(* Logix 5000 project; controller DAD143_Test0 1769-L16ER-BB1B rev 34.12; software revision 34.01; part 2 of 2 *)
(* tags used below, declared in another part *)
   CE_Write_Done : BOOL;
   Done_CE : BOOL;
   CE_Start : BOOL;
   Cycle_Start : BOOL;
   DecimalPoint : SINT;
   Display_real : REAL;
   DisplayStr : STRING;
   DP : BOOL;
   DP_Cahr : STRING;
   DP_Read_Par : SINT[3];
   DP_Read_Res : SINT[5];
   DP_Val : SINT;
   DpPos : DINT;
   DS : BOOL;
   DS_Change : BOOL;
   DS_Change_Handshake : BOOL;
   DS_Change_Tag : BOOL;
   DS_Read_Par : SINT[3];
   DS_Read_Res : SINT[5];
   DS_Step1 : BOOL;
   DS_Val : DINT;
   FinalStr : STRING;
   FM_Change : BOOL;
   FM_Change_Handshake : BOOL;
   FM_Change_Tag : BOOL;
   FM_Read_Par : SINT[3];
   FM_Step1 : BOOL;
   FM_Val : SINT;
   gross : BOOL;
   Gross_weight : BOOL;
   Int_reading : BOOL;
   MR : BOOL;
   MR_Change : BOOL;
   MR_Change_Handshake : BOOL;
   MR_Change_Tag : BOOL;
   MR_Read_Par : SINT[3];
   MR_Step1 : BOOL;
   MR_Val : SINT;
   Power_T : TIMER[12];
   Power_T0 : TIMER;
   READ_AOI : AOI_DAD_143_Read[18];
   ReadCDP : MESSAGE;
   ReadDS : MESSAGE;
   Stable_Bit : BOOL;
   Start : BOOL;
   Start_Visibility : BOOL;
   T10 : TIMER;
   T11 : TIMER;
   T12 : TIMER;
   T13 : TIMER;
   T14 : TIMER;
   T15 : TIMER;
   T16 : TIMER;
   T17 : TIMER;
   T18 : TIMER;
   T22 : TIMER;
   T23 : TIMER;
   T24 : TIMER;
   T37 : TIMER;
   T38 : TIMER;
   T39 : TIMER;
   T7 : TIMER;
   T8 : TIMER;
   T9 : TIMER;
   Tare_reset : BOOL;
   Tare_Reset_1 : BOOL;
   Tare_reset_Bit : BOOL;
   Tare_set : BOOL;
   Tare_set_Bit : BOOL;
   TN_Change : BOOL;
   TN_Change_Handshake : BOOL;
   TN_Change_Tag : BOOL;
   TN_Read_Par : SINT[3];
   TN_Step1 : BOOL;
   TN_Val : SINT;
   Write_AOI : AOI_DAD_143_Write[12];
   Write_DS_Par : SINT[7];
   Write_FM_Par : SINT[7];
   Write_MR_Par : SINT[7];
   Write_TN_Par : SINT[7];
   Write_ZI_Par : SINT[7];
   Write_ZN_Par : SINT[7];
   WriteDS : MESSAGE;
   WriteFM : MESSAGE;
   WriteMR : MESSAGE;
   WriteTN : MESSAGE;
   WriteZI : MESSAGE;
   WriteZN : MESSAGE;
   Zero_reset : BOOL;
   Zero_Reset_1 : BOOL;
   Zero_reset_Bit : BOOL;
   Zero_set : BOOL;
   Zero_set_Bit : BOOL;
   ZI_Change : BOOL;
   ZI_Change_Handshake : BOOL;
   ZI_Change_Tag : BOOL;
   ZI_Read_Par : SINT[3];
   ZI_Step1 : BOOL;
   ZI_Val : DINT;
   ZN_Change : BOOL;
   ZN_Change_Handshake : BOOL;
   ZN_Change_Tag : BOOL;
   ZN_Read_Par : SINT[3];
   ZN_Step1 : BOOL;
   ZN_Val : SINT;
(* MainProgram, continued *)

ROUTINE Dispaly_Tare_Zero   (* ladder *)
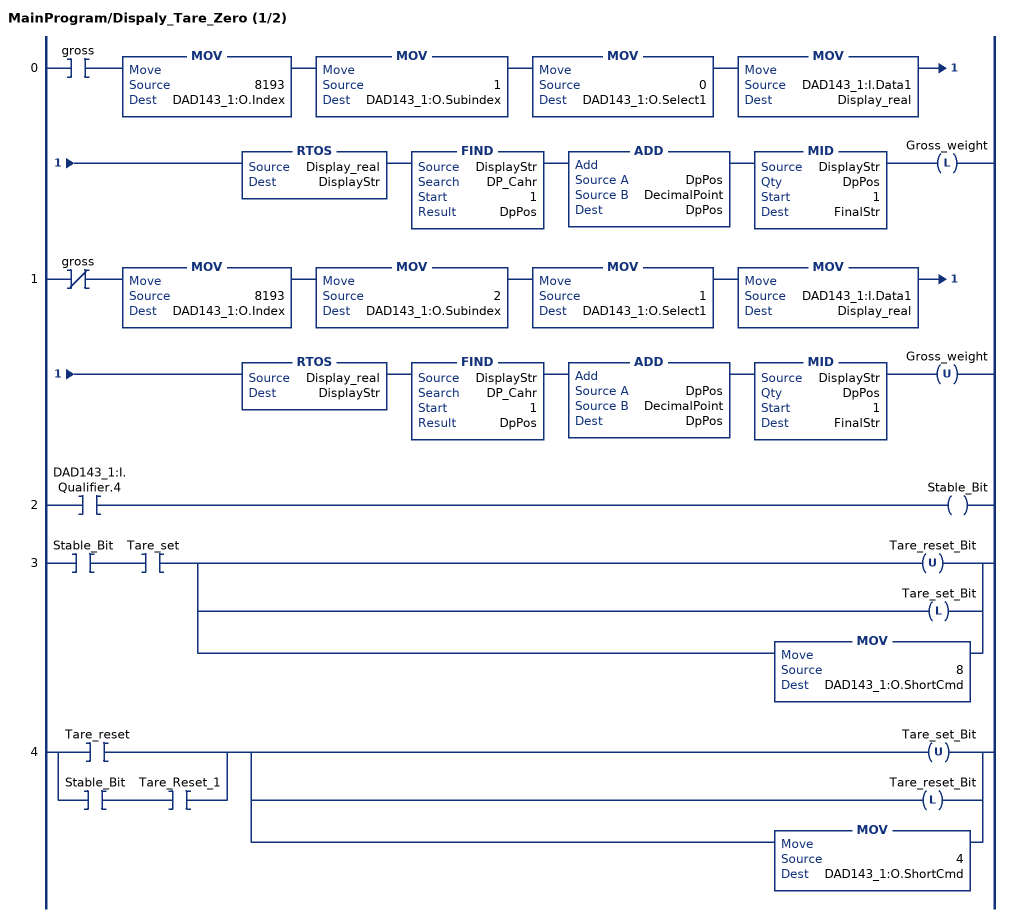
   0: XIC(gross)MOV(8193,DAD143_1:O.Index)MOV(1,DAD143_1:O.Subindex)MOV(0,DAD143_1:O.Select1)MOV(DAD143_1:I.Data1,Display_real)RTOS(Display_real,DisplayStr)FIND(DisplayStr,DP_Cahr,1,DpPos)ADD(DpPos,DecimalPoint,DpPos)MID(DisplayStr,DpPos,1,FinalStr)OTL(Gross_weight);
   1: XIO(gross)MOV(8193,DAD143_1:O.Index)MOV(2,DAD143_1:O.Subindex)MOV(1,DAD143_1:O.Select1)MOV(DAD143_1:I.Data1,Display_real)RTOS(Display_real,DisplayStr)FIND(DisplayStr,DP_Cahr,1,DpPos)ADD(DpPos,DecimalPoint,DpPos)MID(DisplayStr,DpPos,1,FinalStr)OTU(Gross_weight);
   2: XIC(DAD143_1:I.Qualifier.4)OTE(Stable_Bit);
   3: XIC(Stable_Bit)XIC(Tare_set)[[OTU(Tare_reset_Bit) ,OTL(Tare_set_Bit) ] ,MOV(8,DAD143_1:O.ShortCmd) ];
   4: [XIC(Tare_reset) ,XIC(Stable_Bit) XIC(Tare_Reset_1) ][[OTU(Tare_set_Bit) ,OTL(Tare_reset_Bit) ] ,MOV(4,DAD143_1:O.ShortCmd) ];
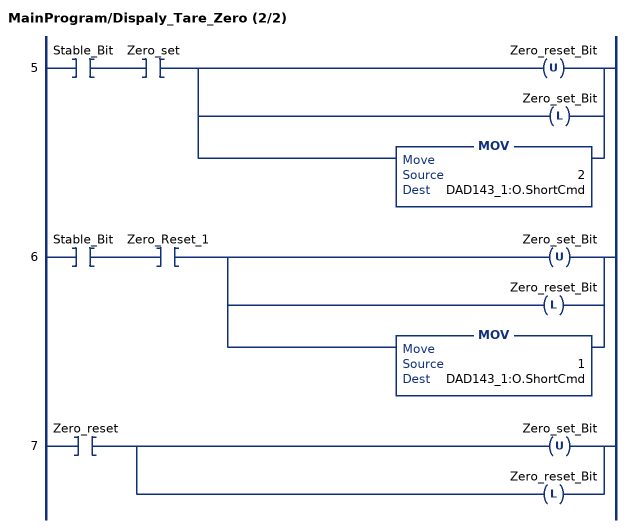
   5: XIC(Stable_Bit)XIC(Zero_set)[[OTU(Zero_reset_Bit) ,OTL(Zero_set_Bit) ] ,MOV(2,DAD143_1:O.ShortCmd) ];
   6: XIC(Stable_Bit)XIC(Zero_Reset_1)[[OTU(Zero_set_Bit) ,OTL(Zero_reset_Bit) ] ,MOV(1,DAD143_1:O.ShortCmd) ];
   7: XIC(Zero_reset)[OTU(Zero_set_Bit) ,OTL(Zero_reset_Bit) ];
END_ROUTINE

ROUTINE Display_Step   (* ladder *)
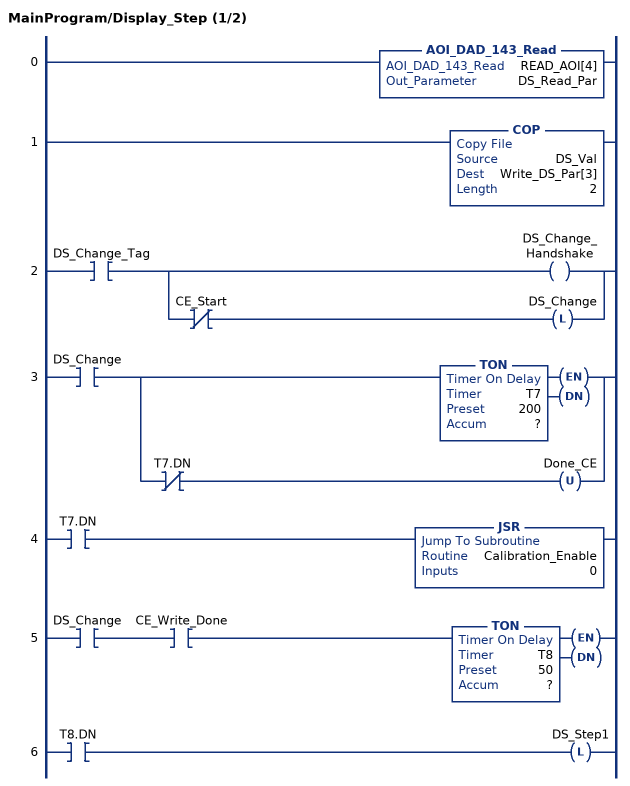
   0: AOI_DAD_143_Read(READ_AOI[4],DS_Read_Par);
   1: COP(DS_Val,Write_DS_Par[3],2);
   2: XIC(DS_Change_Tag)[OTE(DS_Change_Handshake) ,XIO(CE_Start) OTL(DS_Change) ];
   3: XIC(DS_Change)[TON(T7,?,?) ,XIO(T7.DN) OTU(Done_CE) ];
   4: XIC(T7.DN)JSR(Calibration_Enable,0);
   5: XIC(DS_Change)XIC(CE_Write_Done)TON(T8,?,?);
   6: XIC(T8.DN)OTL(DS_Step1);
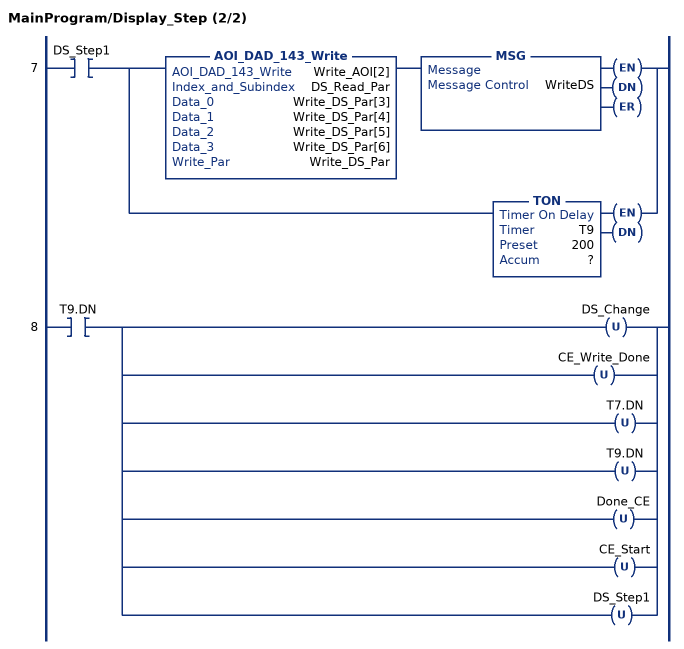
   7: XIC(DS_Step1)[AOI_DAD_143_Write(Write_AOI[2],DS_Read_Par,Write_DS_Par[3],Write_DS_Par[4],Write_DS_Par[5],Write_DS_Par[6],Write_DS_Par) MSG(WriteDS) ,TON(T9,?,?) ];
   8: XIC(T9.DN)[OTU(DS_Change) ,OTU(CE_Write_Done) ,OTU(T7.DN) ,OTU(T9.DN) ,OTU(Done_CE) ,OTU(CE_Start) ,OTU(DS_Step1) ];
END_ROUTINE

ROUTINE Firmware   (* ladder *)
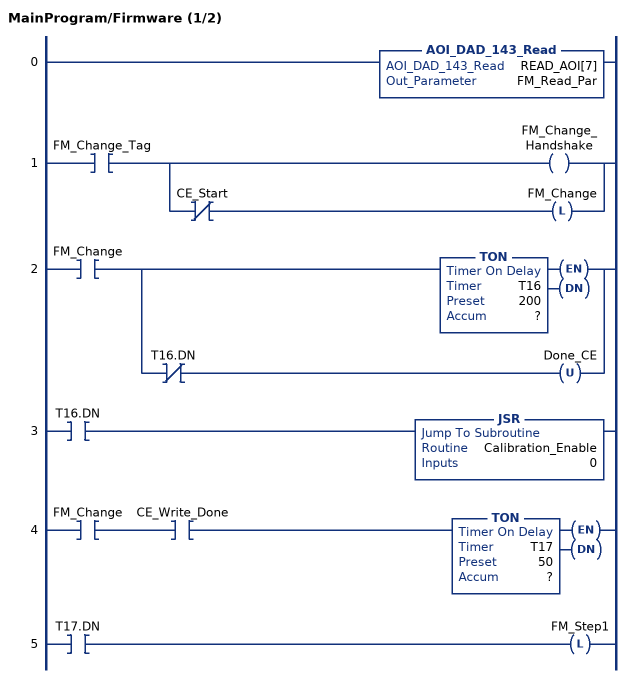
   0: AOI_DAD_143_Read(READ_AOI[7],FM_Read_Par);
   1: XIC(FM_Change_Tag)[OTE(FM_Change_Handshake) ,XIO(CE_Start) OTL(FM_Change) ];
   2: XIC(FM_Change)[TON(T16,?,?) ,XIO(T16.DN) OTU(Done_CE) ];
   3: XIC(T16.DN)JSR(Calibration_Enable,0);
   4: XIC(FM_Change)XIC(CE_Write_Done)TON(T17,?,?);
   5: XIC(T17.DN)OTL(FM_Step1);
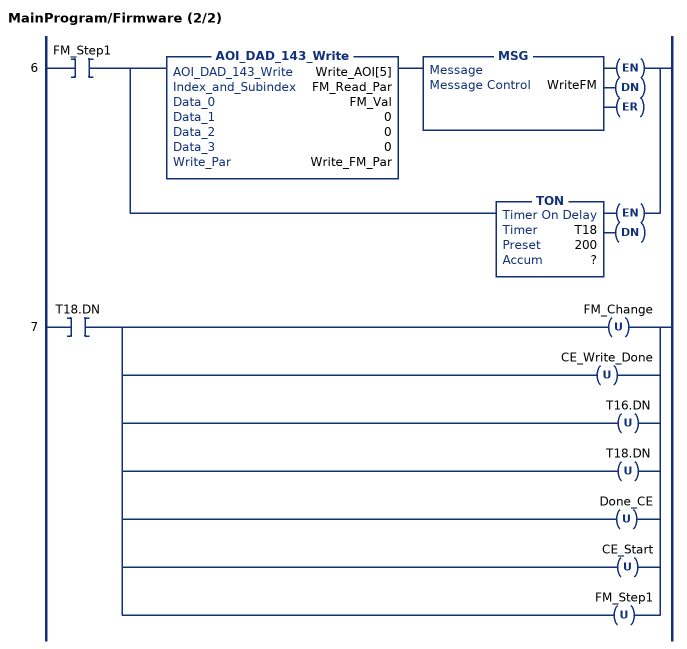
   6: XIC(FM_Step1)[AOI_DAD_143_Write(Write_AOI[5],FM_Read_Par,FM_Val,0,0,0,Write_FM_Par) MSG(WriteFM) ,TON(T18,?,?) ];
   7: XIC(T18.DN)[OTU(FM_Change) ,OTU(CE_Write_Done) ,OTU(T16.DN) ,OTU(T18.DN) ,OTU(Done_CE) ,OTU(CE_Start) ,OTU(FM_Step1) ];
END_ROUTINE

ROUTINE MainRoutine   (* ladder *)
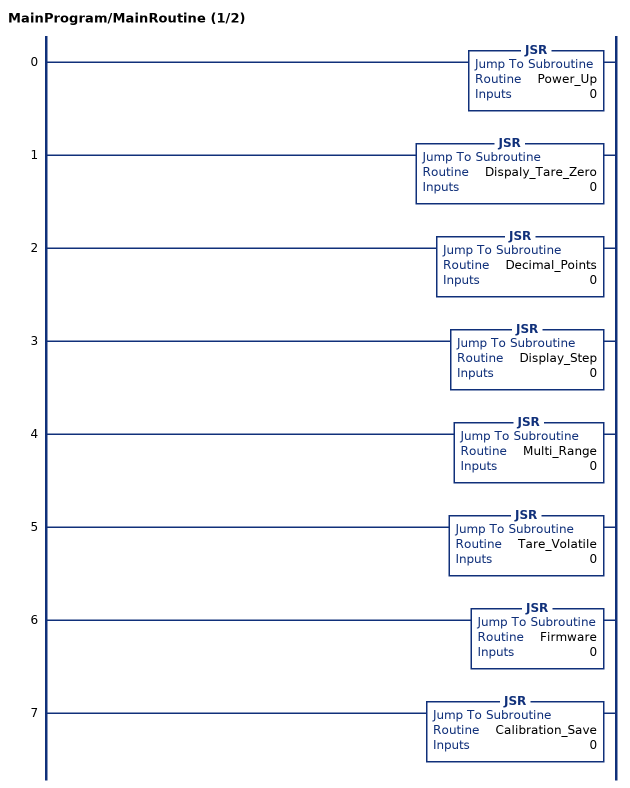
   0: JSR(Power_Up,0);
   1: JSR(Dispaly_Tare_Zero,0);
   2: JSR(Decimal_Points,0);
   3: JSR(Display_Step,0);
   4: JSR(Multi_Range,0);
   5: JSR(Tare_Volatile,0);
   6: JSR(Firmware,0);
   7: JSR(Calibration_Save,0);
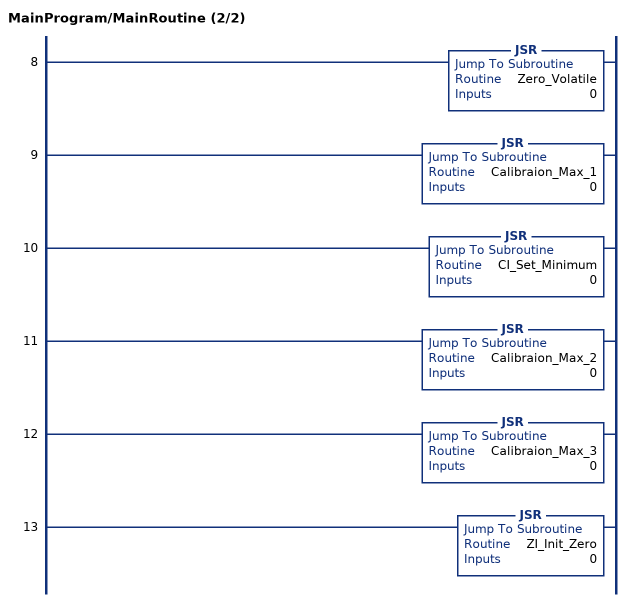
   8: JSR(Zero_Volatile,0);
   9: JSR(Calibraion_Max_1,0);
   10: JSR(CI_Set_Minimum,0);
   11: JSR(Calibraion_Max_2,0);
   12: JSR(Calibraion_Max_3,0);
   13: JSR(ZI_Init_Zero,0);
END_ROUTINE

ROUTINE Multi_Range   (* ladder *)
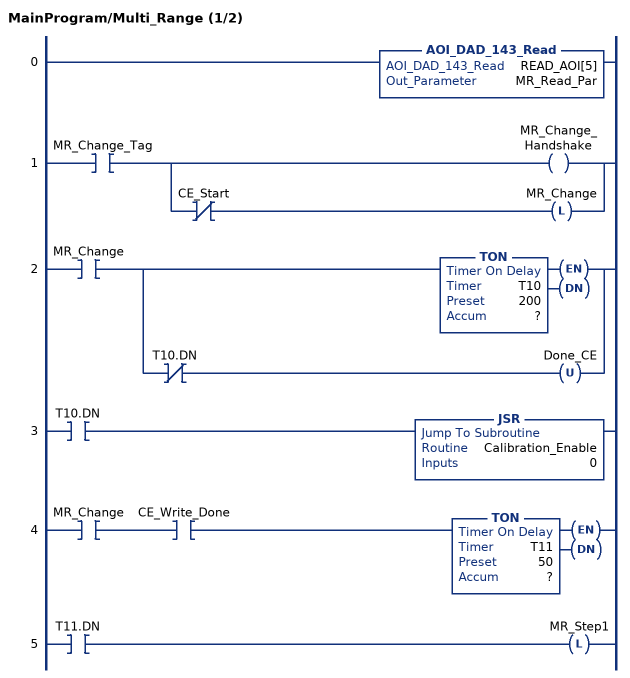
   0: AOI_DAD_143_Read(READ_AOI[5],MR_Read_Par);
   1: XIC(MR_Change_Tag)[OTE(MR_Change_Handshake) ,XIO(CE_Start) OTL(MR_Change) ];
   2: XIC(MR_Change)[TON(T10,?,?) ,XIO(T10.DN) OTU(Done_CE) ];
   3: XIC(T10.DN)JSR(Calibration_Enable,0);
   4: XIC(MR_Change)XIC(CE_Write_Done)TON(T11,?,?);
   5: XIC(T11.DN)OTL(MR_Step1);
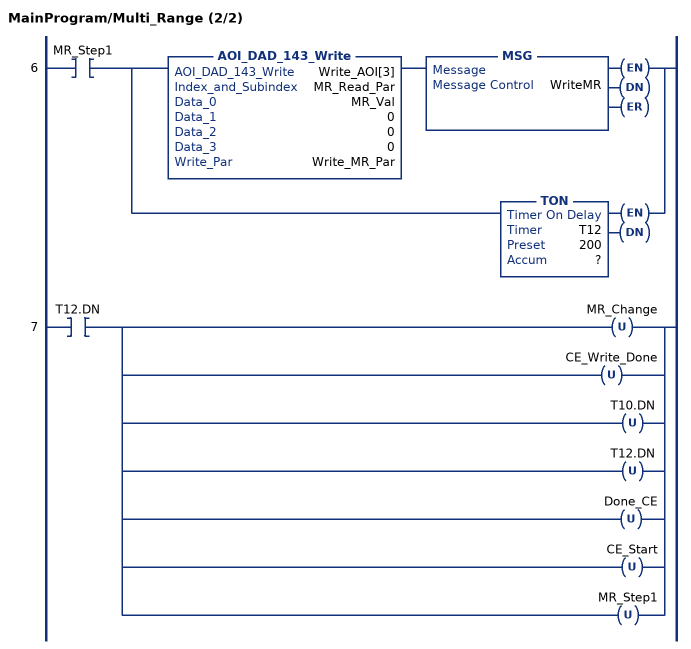
   6: XIC(MR_Step1)[AOI_DAD_143_Write(Write_AOI[3],MR_Read_Par,MR_Val,0,0,0,Write_MR_Par) MSG(WriteMR) ,TON(T12,?,?) ];
   7: XIC(T12.DN)[OTU(MR_Change) ,OTU(CE_Write_Done) ,OTU(T10.DN) ,OTU(T12.DN) ,OTU(Done_CE) ,OTU(CE_Start) ,OTU(MR_Step1) ];
END_ROUTINE

ROUTINE Power_Up   (* ladder *)
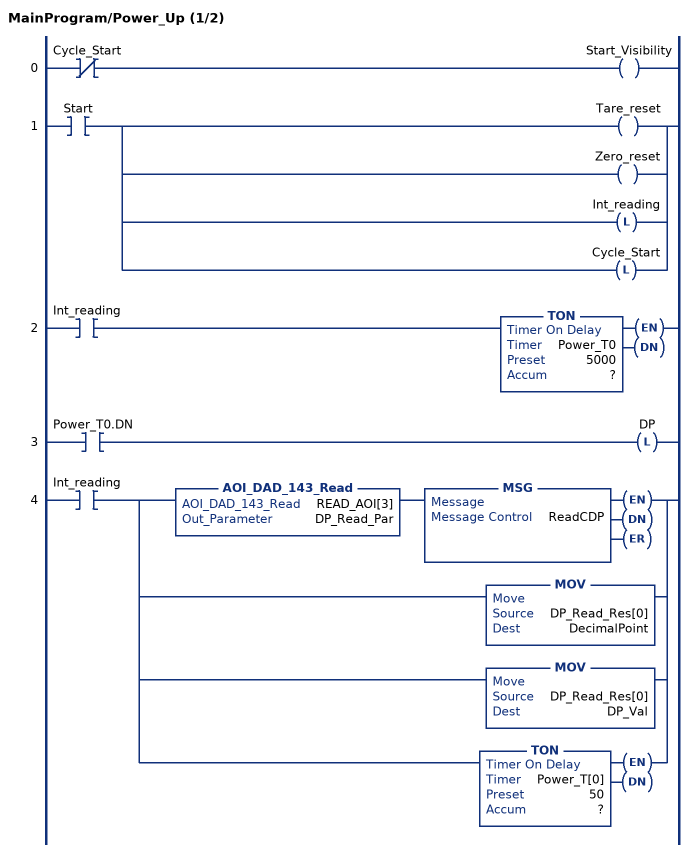
   0: XIO(Cycle_Start)OTE(Start_Visibility);
   1: XIC(Start)[OTE(Tare_reset) ,OTE(Zero_reset) ,OTL(Int_reading) ,OTL(Cycle_Start) ];
   2: XIC(Int_reading)TON(Power_T0,?,?);
   3: XIC(Power_T0.DN)OTL(DP);
   4: XIC(Int_reading)[AOI_DAD_143_Read(READ_AOI[3],DP_Read_Par) MSG(ReadCDP) ,MOV(DP_Read_Res[0],DecimalPoint) ,MOV(DP_Read_Res[0],DP_Val) ,TON(Power_T[0],?,?) ];
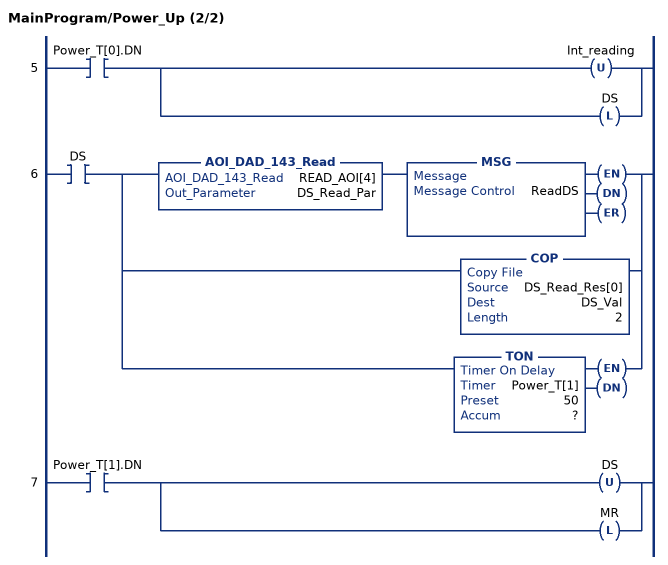
   5: XIC(Power_T[0].DN)[OTU(Int_reading) ,OTL(DS) ];
   6: XIC(DS)[AOI_DAD_143_Read(READ_AOI[4],DS_Read_Par) MSG(ReadDS) ,COP(DS_Read_Res[0],DS_Val,2) ,TON(Power_T[1],?,?) ];
   7: XIC(Power_T[1].DN)[OTU(DS) ,OTL(MR) ];
END_ROUTINE

ROUTINE Tare_Volatile   (* ladder *)
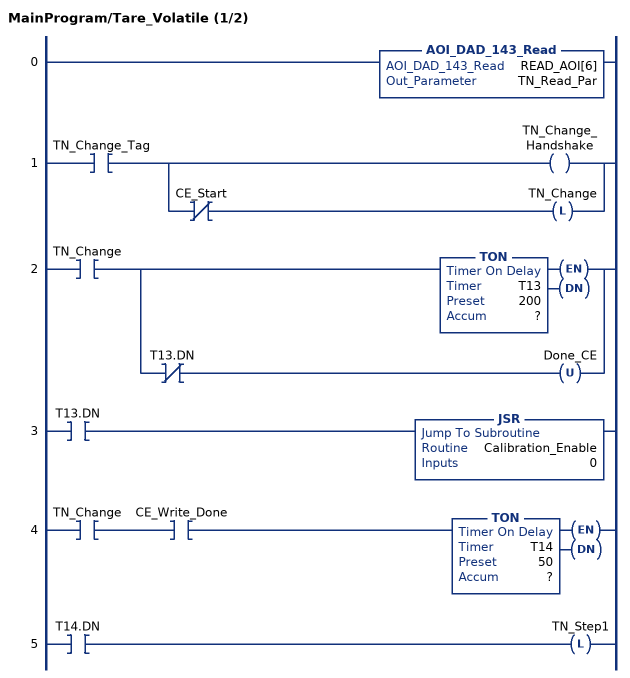
   0: AOI_DAD_143_Read(READ_AOI[6],TN_Read_Par);
   1: XIC(TN_Change_Tag)[OTE(TN_Change_Handshake) ,XIO(CE_Start) OTL(TN_Change) ];
   2: XIC(TN_Change)[TON(T13,?,?) ,XIO(T13.DN) OTU(Done_CE) ];
   3: XIC(T13.DN)JSR(Calibration_Enable,0);
   4: XIC(TN_Change)XIC(CE_Write_Done)TON(T14,?,?);
   5: XIC(T14.DN)OTL(TN_Step1);
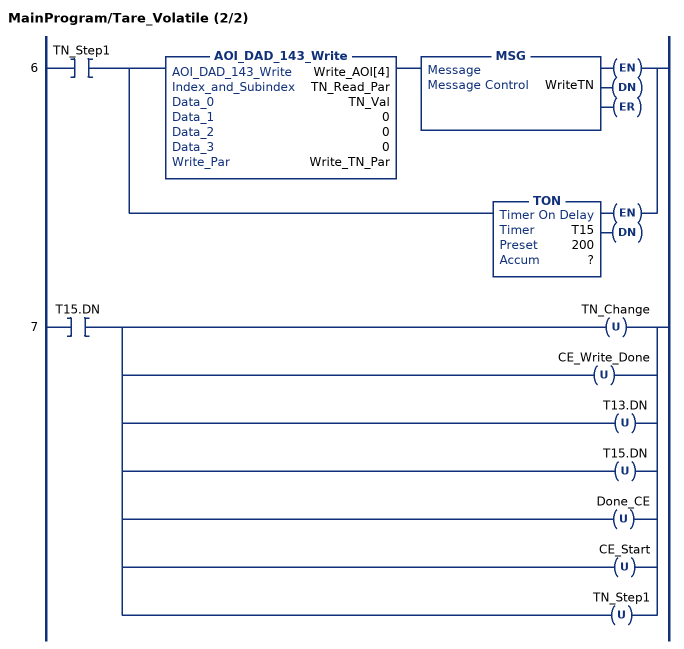
   6: XIC(TN_Step1)[AOI_DAD_143_Write(Write_AOI[4],TN_Read_Par,TN_Val,0,0,0,Write_TN_Par) MSG(WriteTN) ,TON(T15,?,?) ];
   7: XIC(T15.DN)[OTU(TN_Change) ,OTU(CE_Write_Done) ,OTU(T13.DN) ,OTU(T15.DN) ,OTU(Done_CE) ,OTU(CE_Start) ,OTU(TN_Step1) ];
END_ROUTINE

ROUTINE Zero_Volatile   (* ladder *)
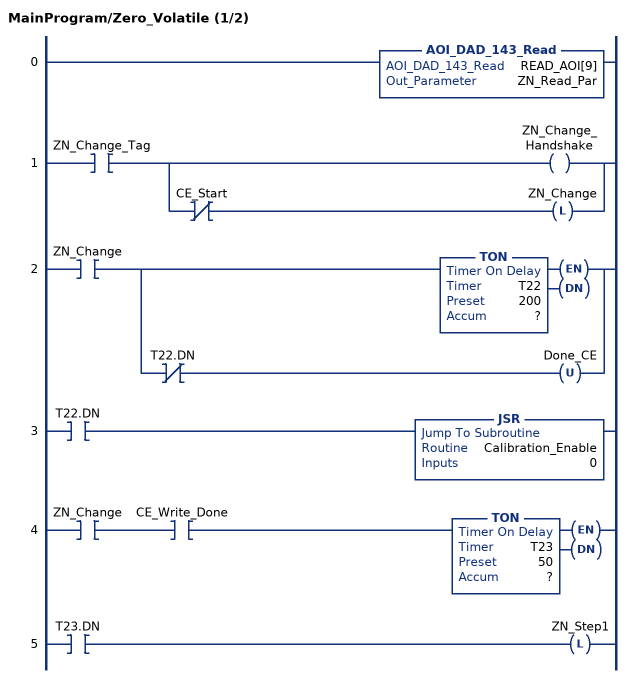
   0: AOI_DAD_143_Read(READ_AOI[9],ZN_Read_Par);
   1: XIC(ZN_Change_Tag)[OTE(ZN_Change_Handshake) ,XIO(CE_Start) OTL(ZN_Change) ];
   2: XIC(ZN_Change)[TON(T22,?,?) ,XIO(T22.DN) OTU(Done_CE) ];
   3: XIC(T22.DN)JSR(Calibration_Enable,0);
   4: XIC(ZN_Change)XIC(CE_Write_Done)TON(T23,?,?);
   5: XIC(T23.DN)OTL(ZN_Step1);
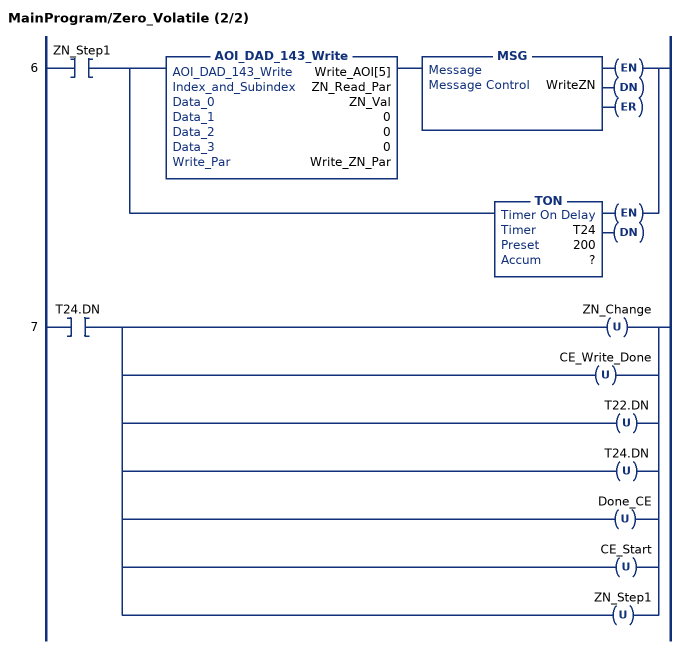
   6: XIC(ZN_Step1)[AOI_DAD_143_Write(Write_AOI[5],ZN_Read_Par,ZN_Val,0,0,0,Write_ZN_Par) MSG(WriteZN) ,TON(T24,?,?) ];
   7: XIC(T24.DN)[OTU(ZN_Change) ,OTU(CE_Write_Done) ,OTU(T22.DN) ,OTU(T24.DN) ,OTU(Done_CE) ,OTU(CE_Start) ,OTU(ZN_Step1) ];
END_ROUTINE

ROUTINE ZI_Init_Zero   (* ladder *)
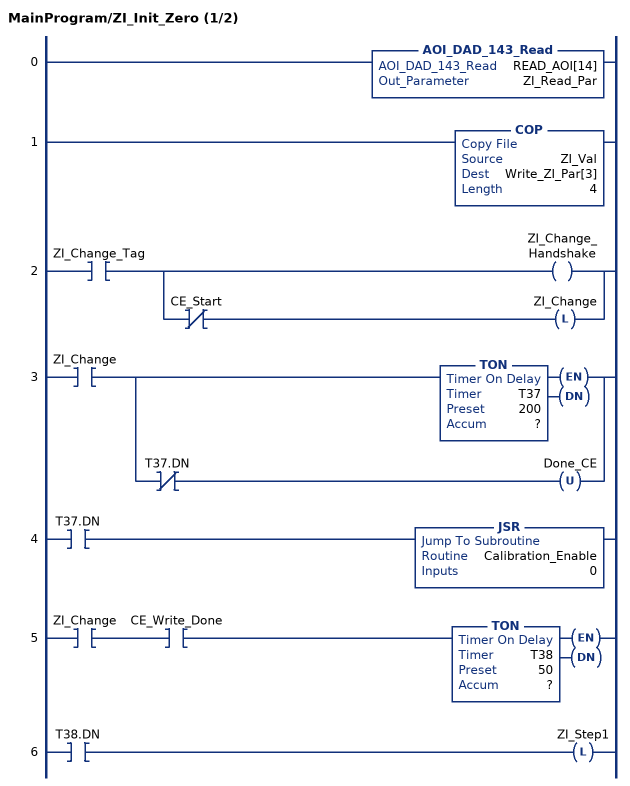
   0: AOI_DAD_143_Read(READ_AOI[14],ZI_Read_Par);
   1: COP(ZI_Val,Write_ZI_Par[3],4);
   2: XIC(ZI_Change_Tag)[OTE(ZI_Change_Handshake) ,XIO(CE_Start) OTL(ZI_Change) ];
   3: XIC(ZI_Change)[TON(T37,?,?) ,XIO(T37.DN) OTU(Done_CE) ];
   4: XIC(T37.DN)JSR(Calibration_Enable,0);
   5: XIC(ZI_Change)XIC(CE_Write_Done)TON(T38,?,?);
   6: XIC(T38.DN)OTL(ZI_Step1);
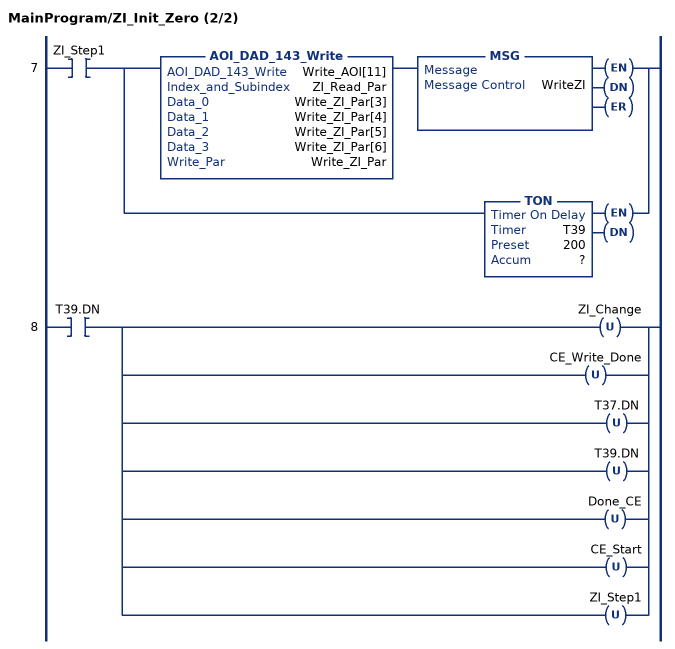
   7: XIC(ZI_Step1)[AOI_DAD_143_Write(Write_AOI[11],ZI_Read_Par,Write_ZI_Par[3],Write_ZI_Par[4],Write_ZI_Par[5],Write_ZI_Par[6],Write_ZI_Par) MSG(WriteZI) ,TON(T39,?,?) ];
   8: XIC(T39.DN)[OTU(ZI_Change) ,OTU(CE_Write_Done) ,OTU(T37.DN) ,OTU(T39.DN) ,OTU(Done_CE) ,OTU(CE_Start) ,OTU(ZI_Step1) ];
END_ROUTINE
END_PROGRAM
